// TIA Portal V20 export
FUNCTION_BLOCK "FB_DigitalInputsSonplas"   // FB211, SCL
{ S7_Optimized_Access := 'TRUE' }
// stored: AutoNumber false, MemoryReserve 100, SetENOAutomatically false
   VAR
      sSonplasDiagDPCoupler { S7_SetPoint := 'True'} : "FB_DigitalInput";
      sSonplasReady { S7_SetPoint := 'True'} : "FB_DigitalInput";
      sSonplasNoEStop { S7_SetPoint := 'True'} : "FB_DigitalInput";
      sSonplasDoorsClosed { S7_SetPoint := 'True'} : "FB_DigitalInput";
      sSonplasRunError { S7_SetPoint := 'True'} : "FB_DigitalInput";
      sSonplasFreeI200_5 { S7_SetPoint := 'True'} : "FB_DigitalInput";
      sSonplasFreeI200_6 { S7_SetPoint := 'True'} : "FB_DigitalInput";
      sSonplasFreeI200_7 { S7_SetPoint := 'True'} : "FB_DigitalInput";
      sSonplasFreeI201_0 { S7_SetPoint := 'True'} : "FB_DigitalInput";
      sSonplasOutCollision { S7_SetPoint := 'True'} : "FB_DigitalInput";
      sSonplasFreeI201_2 { S7_SetPoint := 'True'} : "FB_DigitalInput";
      Sonpla_FreeI201_3 { S7_SetPoint := 'True'} : "FB_DigitalInput";
      sSonplasFreeI201_4 { S7_SetPoint := 'True'} : "FB_DigitalInput";
      sSonplasFreeI201_5 { S7_SetPoint := 'True'} : "FB_DigitalInput";
      sSonplasFreeI201_6 { S7_SetPoint := 'True'} : "FB_DigitalInput";
      sSonplasFreeI201_7 { S7_SetPoint := 'True'} : "FB_DigitalInput";
      sSonplasShuttle1Finished { S7_SetPoint := 'True'} : "FB_DigitalInput";
      sSonplasFreeI202_1 { S7_SetPoint := 'True'} : "FB_DigitalInput";
      sSonplasFreeI202_2 { S7_SetPoint := 'True'} : "FB_DigitalInput";
      sSonplasFreeI202_3 { S7_SetPoint := 'True'} : "FB_DigitalInput";
      sSonplasFreeI202_4 { S7_SetPoint := 'True'} : "FB_DigitalInput";
      sSonplasFreeI202_5 { S7_SetPoint := 'True'} : "FB_DigitalInput";
      sSonplasFreeI202_6 { S7_SetPoint := 'True'} : "FB_DigitalInput";
      sSonplasFreeI202_7 { S7_SetPoint := 'True'} : "FB_DigitalInput";
      sSonplasShuttle2Finished { S7_SetPoint := 'True'} : "FB_DigitalInput";
      sSonplasFreeI203_1 { S7_SetPoint := 'True'} : "FB_DigitalInput";
      sSonplasFreeI203_2 { S7_SetPoint := 'True'} : "FB_DigitalInput";
      sSonplasFreeI203_3 { S7_SetPoint := 'True'} : "FB_DigitalInput";
      sSonplasFreeI203_4 { S7_SetPoint := 'True'} : "FB_DigitalInput";
      sSonplasFreeI203_5 { S7_SetPoint := 'True'} : "FB_DigitalInput";
      sSonplasFreeI203_6 { S7_SetPoint := 'True'} : "FB_DigitalInput";
      sSonplasFreeI203_7 { S7_SetPoint := 'True'} : "FB_DigitalInput";
      sSonplasFlowResultAvail { S7_SetPoint := 'True'} : "FB_DigitalInput";
      sSonplasFreeI244_1 { S7_SetPoint := 'True'} : "FB_DigitalInput";
      sSonplasFreeI244_2 { S7_SetPoint := 'True'} : "FB_DigitalInput";
      sSonplasFreeI244_3 { S7_SetPoint := 'True'} : "FB_DigitalInput";
      sSonplasFreeI244_4 { S7_SetPoint := 'True'} : "FB_DigitalInput";
      sSonplasFreeI244_5 { S7_SetPoint := 'True'} : "FB_DigitalInput";
      sSonplasFreeI244_6 { S7_SetPoint := 'True'} : "FB_DigitalInput";
      sSonplasFreeI244_7 { S7_SetPoint := 'True'} : "FB_DigitalInput";
   END_VAR
BEGIN
   REGION Description head
       //==================================================================================
       // POSALUX Swiss SA / (C) Copyright 2025
       //----------------------------------------------------------------------------------
       // Title: Digital Inputs mapping
       // Comment/Function: Sonplas Digital Inputs mapping
       // Author: Fabien WALDT
       // Engineering: TIA Portal v17
       //----------------------------------------------------------------------------------
       // Change log table:
       // Version  | Date     | Expert in charge | Changes applied
       // ---------|----------|------------------|-----------------------------------------
       // 00.00.01 | 20250423 | WFA              | First released version
       // =================================================================================
   END_REGION


   REGION Operating modes and parts exchange
       #sSonplasDiagDPCoupler(iHWStatus := "DI_SonplasDiagDPCoupler");
       #sSonplasReady(iHWStatus := "DI_SonplasReady");
       #sSonplasNoEStop(iHWStatus := "DI_SonplasNoEStop");
       #sSonplasDoorsClosed(iHWStatus := "DI_SonplasDoorsClosed");
       #sSonplasRunError(iHWStatus := "DI_SonplasRunError");
       #sSonplasFreeI200_5(iHWStatus := "DI_SonplasFreeI200_5");
       #sSonplasFreeI200_6(iHWStatus := "DI_SonplasFreeI200_6");
       #sSonplasFreeI200_7(iHWStatus := "DI_SonplasFreeI200_7");
       // 
       #sSonplasFreeI201_0(iHWStatus := "DI_SonplasFreeI201_0");
       #sSonplasOutCollision(iHWStatus := "DI_SonplasOutCollision");
       #sSonplasFreeI201_2(iHWStatus := "DI_SonplasFreeI201_2");
       #Sonpla_FreeI201_3(iHWStatus := "DI_SonplasFreeI201_3");
       #sSonplasFreeI201_4(iHWStatus := "DI_SonplasFreeI201_4");
       #sSonplasFreeI201_5(iHWStatus := "DI_SonplasFreeI201_5");
       #sSonplasFreeI201_6(iHWStatus := "DI_SonplasFreeI201_6");
       #sSonplasFreeI201_7(iHWStatus := "DI_SonplasFreeI201_7");
   END_REGION

   REGION Part exchange
       #sSonplasShuttle1Finished(iHWStatus := "DI_SonplasShuttle1Finished");
       #sSonplasFreeI202_1(iHWStatus := "DI_SonplasFreeI202_1");
       #sSonplasFreeI202_2(iHWStatus := "DI_SonplasFreeI202_2");
       #sSonplasFreeI202_3(iHWStatus := "DI_SonplasFreeI202_3");
       #sSonplasFreeI202_4(iHWStatus := "DI_SonplasFreeI202_4");
       #sSonplasFreeI202_5(iHWStatus := "DI_SonplasFreeI202_5");
       #sSonplasFreeI202_6(iHWStatus := "DI_SonplasFreeI202_6");
       #sSonplasFreeI202_7(iHWStatus := "DI_SonplasFreeI202_7");
       //
       #sSonplasShuttle2Finished(iHWStatus := "DI_SonplasShuttle2Finished");
       #sSonplasFreeI203_1(iHWStatus := "DI_SonplasFreeI203_1");
       #sSonplasFreeI203_2(iHWStatus := "DI_SonplasFreeI203_2");
       #sSonplasFreeI203_3(iHWStatus := "DI_SonplasFreeI203_3");
       #sSonplasFreeI203_4(iHWStatus := "DI_SonplasFreeI203_4");
       #sSonplasFreeI203_5(iHWStatus := "DI_SonplasFreeI203_5");
       #sSonplasFreeI203_6(iHWStatus := "DI_SonplasFreeI203_6");
       #sSonplasFreeI203_7(iHWStatus := "DI_SonplasFreeI203_7");
   END_REGION

   REGION Measure
       #sSonplasFlowResultAvail(iHWStatus := "DI_SonplasFlowResultAvail");
       #sSonplasFreeI244_1(iHWStatus := "DI_SonplasFreeI244_1");
       #sSonplasFreeI244_2(iHWStatus := "DI_SonplasFreeI244_2");
       #sSonplasFreeI244_3(iHWStatus := "DI_SonplasFreeI244_3");
       #sSonplasFreeI244_4(iHWStatus := "DI_SonplasFreeI244_4");
       #sSonplasFreeI244_5(iHWStatus := "DI_SonplasFreeI244_5");
       #sSonplasFreeI244_6(iHWStatus := "DI_SonplasFreeI244_6");
       #sSonplasFreeI244_7(iHWStatus := "DI_SonplasFreeI244_7");
   END_REGION
END_FUNCTION_BLOCK
